(* IEC 61131-3 sources: com.logicals.lc3.webinar/usRTS_RPMControl_iSOC/src_FB_LIB_SAFE/Compare/BOOL, 2 files *)

(* ---- wEQ_BOOL_2.iecst ---- *)
NAMESPACE logicals.web.standard
NAMESPACE compare

/*
 * Function block wrapper for IEC 61131-3 EQ<br>
 * IN1 =  1st value (BOOL)<br>
 * IN2 =  2nd value (BOOL)<br>
 * OUT = true if IN1 is equal to IN2 (BOOL)<br>
 */
FUNCTION_BLOCK wEQ_BOOL_2
	{ vNameAlignment:="center"; altName:="="; bgColor:="MediumBlue"; width:=40; hideIONames; }
	VAR_INPUT
		IN1 : BOOL;
		IN2 : BOOL;
	END_VAR
	VAR_OUTPUT
		OUT : BOOL;
	END_VAR

	OUT := EQ(IN1:=IN1, IN2:=IN2, ENO=>ENO);
END_FUNCTION_BLOCK

END_NAMESPACE
END_NAMESPACE

(* ---- wNE_BOOL.iecst ---- *)
NAMESPACE logicals.web.standard
NAMESPACE compare

/*
 * Function block wrapper for IEC 61131-3 NE<br>
 * IN1 = value 1 (BOOL)<br>
 * IN2 = value 2 (BOOL)<br>
 * OUT = true if IN1 is not equal to IN2 (BOOL)<br>
 */
FUNCTION_BLOCK wNE_BOOL
	{ vNameAlignment:="center"; altName:="<>"; bgColor:="MediumBlue"; width:=40; hideIONames; }
	VAR_INPUT
		IN1 : BOOL;
		IN2 : BOOL;
	END_VAR
	VAR_OUTPUT
		OUT : BOOL;
	END_VAR

	OUT := NE(IN1:=IN1, IN2:=IN2, ENO=>ENO);
END_FUNCTION_BLOCK

END_NAMESPACE
END_NAMESPACE
